# B&R Automation Studio project Model-repo
Automation Studio 4.5.2.102

## Configuration PLC

CPU X20CP1586, AutomationRuntime G4.53, Build 4.1.2, Vc V4.52.0

### Hardware
```
X20CP1586 : X20CP1586 v1.5.0.0
  Connector IF2:
    ActivateDevice = 1
    Mode = Manual
    InternetAddress = 192.168.0.5
    SubnetMask = 255.255.255.0
  Connector IF3:
    Operation = EthOnly
  ConfigurationID = JS_PLC
  ActivateOpcUa = 1
  OpcUaActivateAuditEvents = 1
  OpcUa_AuthenticationSecurityPolicy_EnableNone = 1
  OpcUa_AuthenticationSecurityPolicy_EnableBasic128Rsa15 = 1
  OpcUaInformationModels_PV_Version = 1
```

## Logical view

### Program Logical/Model/pend_mod

#### pend_mod.c
```c
/********************************************************************
 * COPYRIGHT -- Bernecker + Rainer Industrie-Elektronik Ges.m.b.H.
 ********************************************************************
 * Program: pend_mod_nlin
 * File: pend_mod.c
 * Author: Bernecker + Rainer Industrie Elektronik Ges.m.b.H.
 * Created: Fri Apr 16 22:40:22 2010
 ********************************************************************
 * Implementation of program pend_mod_nlin
 ********************************************************************
 * Generated with B&R Automation Studio Target for Simulink  V6.1.0
 * (ERT based)
 ********************************************************************/

#define _ASMATH_
#define ASMATH_
#define _ASMATH_H
#define ASMATH_H
#define _ASMATH_H_
#define ASMATH_H_
#define _ASSTRING_
#define ASSTRING_
#define _ASSTRING_H
#define ASSTRING_H
#define _ASSTRING_H_
#define ASSTRING_H_
#include <bur/plctypes.h>
#ifdef _DEFAULT_INCLUDES
#include <AsDefault.h>
#endif

#include "pend_mod_nlin.h"
#include "rtwtypes.h"

/*  Defines */

/*  Data Types */

/**************************** GLOBAL DATA *************************************/
/*  Definitions */

/*  Declarations  */

/***************************** FILE SCOPE DATA ********************************/

/*************************** FUNCTIONS ****************************************/
#ifdef __cplusplus

unsigned long bur_heap_size = 6553500;

#endif

  void _INIT mainINIT(void)
{

    UDINT st_ident;
  RTInfo_typ rt_info;
  rt_info.enable = 1;
  RTInfo(&rt_info);
  if (rt_info.cycle_time != 10000) {
    /* cycle time does not match Simulink fixed-step size */
    ST_ident("pend_mod", 0, &st_ident);
    ST_tmp_suspend(st_ident);
    ERR_warning(33310, 0);
  }

  /* initialize model */
  pend_mod_nlin_initialize();

} void _CYCLIC mainCYCLIC(void)
{
	if(start)
	{/* call model step function */
		pend_mod_nlin_output();
		pend_mod_nlin_update();
	}
	if(reset)
	{
		start = 0;
		pend_mod_nlin_initialize();
		ref = 0;
		x[0] = x[1] = x[2] = x[3] = 0;
		y[0] = y[1] = 0;
		F = 0;
		reset = 0;
	}
}  void _EXIT mainEXIT(void)
{
  /* terminate model */
  pend_mod_nlin_terminate();

} /*****************************************************************************
     Task sample time: 0.01s
   *****************************************************************************/
/*****************************************************************************
   B&R Automation Studio Target for Simulink Version: V6.1.0 (06-Nov-2019)
 *****************************************************************************/

/*======================== TOOL VERSION INFORMATION ==========================*
 * MATLAB 9.7 (R2019b)18-Jul-2019                                             *
 * Simulink 10.0 (R2019b)18-Jul-2019                                          *
 * Simulink Coder 9.2 (R2019b)18-Jul-2019                                     *
 * Embedded Coder 7.3 (R2019b)18-Jul-2019                                     *
 * Stateflow 10.1 (R2019b)18-Jul-2019                                         *
 * Fixed-Point Designer 6.4 (R2019b)18-Jul-2019                               *
 *============================================================================*/

/*======================= LICENSE IN USE INFORMATION =========================*
 * control_toolbox                                                            *
 * matlab                                                                     *
 * matlab_coder                                                               *
 * real-time_workshop                                                         *
 * rtw_embedded_coder                                                         *
 * simulink                                                                   *
 *============================================================================*/
```

### Program Logical/Controller/pend_ctrl

#### pend_ctrl_lin.h
```c
/********************************************************************
 * COPYRIGHT -- Bernecker + Rainer Industrie-Elektronik Ges.m.b.H.
 ********************************************************************
 * Program: pend_ctrl_lin
 * File: pend_ctrl_lin.h
 * Author: Bernecker + Rainer Industrie Elektronik Ges.m.b.H.
 * Created: Wed Mar 17 14:21:47 2010
 ********************************************************************
 * Header for program pend_ctrl_lin
 ********************************************************************
 * Generated with B&R Automation Studio Target for Simulink  V6.1.0
 * (ERT based)
 ********************************************************************/

#ifndef RTW_HEADER_pend_ctrl_lin_h_
#define RTW_HEADER_pend_ctrl_lin_h_
#ifndef pend_ctrl_lin_COMMON_INCLUDES_
# define pend_ctrl_lin_COMMON_INCLUDES_
#include "rtwtypes.h"
#include "rtw_continuous.h"
#include "rtw_solver.h"
#endif                                 /* pend_ctrl_lin_COMMON_INCLUDES_ */

#include <bur/plctypes.h>

#ifdef _DEFAULT_INCLUDES
 #include <AsDefault.h>
#endif

#ifndef AST_ROUND
#define AST_ROUND(x) ((x)>=0?(long long)((x)+0.5):(long long)((x)-0.5))
#endif

#include "pend_ctrl_lin_types.h"

/* Macros for accessing real-time model data structure */
#ifndef rtmGetErrorStatus
# define rtmGetErrorStatus(rtm)        ((rtm)->errorStatus)
#endif

#ifndef rtmSetErrorStatus
# define rtmSetErrorStatus(rtm, val)   ((rtm)->errorStatus = (val))
#endif

#ifndef MIN
#define MIN(a,b)                       ((a) < (b) ? (a) : (b))
#endif

#ifndef MAX
#define MAX(a,b)                       ((a) > (b) ? (a) : (b))
#endif

/* Block signals (default storage) */
typedef struct {
  real_T Input;                        /* '<S1>/Input' */
  real_T ref;                          /* '<Root>/ref' */
  real_T FeedForward;                  /* '<S4>/Feed-Forward' */
  real_T Input_f[4];                   /* '<S3>/Input' */
  real_T LQRController;                /* '<S4>/LQR Controller' */
  real_T Sum;                          /* '<S4>/Sum' */
  real_T Input1[2];                    /* '<S3>/Input1' */
} BlockIO_pend_ctrl_lin;

/* Real-time Model Data Structure */
struct tag_RTM_pend_ctrl_lin {
  const char_T *errorStatus;
};

/* Block signals (default storage) */
extern BlockIO_pend_ctrl_lin pend_ctrl_lin_B;

/* Model entry point functions */
extern void pend_ctrl_lin_initialize(void);
extern void pend_ctrl_lin_output(void);
extern void pend_ctrl_lin_update(void);
extern void pend_ctrl_lin_terminate(void);

/* Real-time Model object */
extern RT_MODEL_pend_ctrl_lin *const pend_ctrl_lin_M;

/*-
 * The generated code includes comments that allow you to trace directly
 * back to the appropriate location in the model.  The basic format
 * is <system>/block_name, where system is the system number (uniquely
 * assigned by Simulink) and block_name is the name of the block.
 *
 * Use the MATLAB hilite_system command to trace the generated code back
 * to the model.  For example,
 *
 * hilite_system('<S3>')    - opens system 3
 * hilite_system('<S3>/Kp') - opens and selects block Kp which resides in S3
 *
 * Here is the system hierarchy for this model
 *
 * '<Root>' : 'pend_ctrl_lin'
 * '<S1>'   : 'pend_ctrl_lin/B&R reference input'
 * '<S2>'   : 'pend_ctrl_lin/Configurable Controller  Subsystem1'
 * '<S3>'   : 'pend_ctrl_lin/inverted_pendulum_IOs'
 * '<S4>'   : 'pend_ctrl_lin/Configurable Controller  Subsystem1/State Feedback Controller (blks)'
 */
#endif                                 /* RTW_HEADER_pend_ctrl_lin_h_ */
```

#### pend_ctrl.c
```c
/********************************************************************
 * COPYRIGHT -- Bernecker + Rainer Industrie-Elektronik Ges.m.b.H.
 ********************************************************************
 * Program: pend_ctrl_lin
 * File: pend_ctrl.c
 * Author: Bernecker + Rainer Industrie Elektronik Ges.m.b.H.
 * Created: Wed Mar 17 14:21:47 2010
 ********************************************************************
 * Implementation of program pend_ctrl_lin
 ********************************************************************
 * Generated with B&R Automation Studio Target for Simulink  V6.1.0
 * (ERT based)
 ********************************************************************/

#define _ASMATH_
#define ASMATH_
#define _ASMATH_H
#define ASMATH_H
#define _ASMATH_H_
#define ASMATH_H_
#define _ASSTRING_
#define ASSTRING_
#define _ASSTRING_H
#define ASSTRING_H
#define _ASSTRING_H_
#define ASSTRING_H_
#include <bur/plctypes.h>
#ifdef _DEFAULT_INCLUDES
#include <AsDefault.h>
#endif

#include "pend_ctrl_lin.h"
#include "rtwtypes.h"

/*  Defines */

/*  Data Types */

/**************************** GLOBAL DATA *************************************/
/*  Definitions */

/*  Declarations  */

/***************************** FILE SCOPE DATA ********************************/

/*************************** FUNCTIONS ****************************************/
#ifdef __cplusplus

unsigned long bur_heap_size = 6553500;

#endif

  void _INIT mainINIT(void)
{

    UDINT st_ident;
  RTInfo_typ rt_info;
  rt_info.enable = 1;
  RTInfo(&rt_info);
  if (rt_info.cycle_time != 10000) {
    /* cycle time does not match Simulink fixed-step size */
    ST_ident("pend_ctrl", 0, &st_ident);
    ST_tmp_suspend(st_ident);
    ERR_warning(33310, 0);
  }

  /* initialize model */
  pend_ctrl_lin_initialize();

} void _CYCLIC mainCYCLIC(void)
{
  /* call model step function */
  pend_ctrl_lin_output();

  pend_ctrl_lin_update();

} void _EXIT mainEXIT(void)
{
  /* terminate model */
  pend_ctrl_lin_terminate();

} /*****************************************************************************
     Task sample time: 0.01s
   *****************************************************************************/
/*****************************************************************************
   B&R Automation Studio Target for Simulink Version: V6.1.0 (06-Nov-2019)
 *****************************************************************************/

/*======================== TOOL VERSION INFORMATION ==========================*
 * MATLAB 9.7 (R2019b)18-Jul-2019                                             *
 * Simulink 10.0 (R2019b)18-Jul-2019                                          *
 * Simulink Coder 9.2 (R2019b)18-Jul-2019                                     *
 * Embedded Coder 7.3 (R2019b)18-Jul-2019                                     *
 * Stateflow 10.1 (R2019b)18-Jul-2019                                         *
 * Fixed-Point Designer 6.4 (R2019b)18-Jul-2019                               *
 *============================================================================*/

/*======================= LICENSE IN USE INFORMATION =========================*
 * control_toolbox                                                            *
 * matlab                                                                     *
 * matlab_coder                                                               *
 * real-time_workshop                                                         *
 * rtw_embedded_coder                                                         *
 * simulink                                                                   *
 *============================================================================*/
```

#### pend_ctrl_lin.c
```c
/********************************************************************
 * COPYRIGHT -- Bernecker + Rainer Industrie-Elektronik Ges.m.b.H.
 ********************************************************************
 * Program: pend_ctrl_lin
 * File: pend_ctrl_lin.c
 * Author: Bernecker + Rainer Industrie Elektronik Ges.m.b.H.
 * Created: Wed Mar 17 14:21:47 2010
 ********************************************************************
 * Implementation of program pend_ctrl_lin
 ********************************************************************
 * Generated with B&R Automation Studio Target for Simulink  V6.1.0
 * (ERT based)
 ********************************************************************/

#include "pend_ctrl_lin.h"
#include "pend_ctrl_lin_private.h"

/*  Defines */

/*  Data Types */

/**************************** GLOBAL DATA *************************************/
/*  Definitions */

/* Block signals (default storage) */
BlockIO_pend_ctrl_lin pend_ctrl_lin_B;

/* Real-time model */
RT_MODEL_pend_ctrl_lin pend_ctrl_lin_M_;
RT_MODEL_pend_ctrl_lin *const pend_ctrl_lin_M = &pend_ctrl_lin_M_;

/*  Declarations  */

/***************************** FILE SCOPE DATA ********************************/

/*************************** FUNCTIONS ****************************************/

/* Model output function */
void pend_ctrl_lin_output(void)
{
  real_T tmp;

  /* S-Function (bur_in): '<S1>/Input' */
  pend_ctrl_lin_B.Input = ref;

  /* Gain: '<Root>/ref' */
  pend_ctrl_lin_B.ref = 10.0 * pend_ctrl_lin_B.Input;

  /* Gain: '<S4>/Feed-Forward' */
  pend_ctrl_lin_B.FeedForward = -2987.4616903679112 * pend_ctrl_lin_B.ref;

  /* S-Function (bur_in): '<S3>/Input' */
  pend_ctrl_lin_B.Input_f[0] = x[0];
  pend_ctrl_lin_B.Input_f[1] = x[1];
  pend_ctrl_lin_B.Input_f[2] = x[2];
  pend_ctrl_lin_B.Input_f[3] = x[3];

  /* Gain: '<S4>/LQR Controller' */
  tmp = -2987.4616903679125 * pend_ctrl_lin_B.Input_f[0];
  tmp += -3740.1178916812455 * pend_ctrl_lin_B.Input_f[1];
  tmp += -32774.860875805127 * pend_ctrl_lin_B.Input_f[2];
  tmp += -7399.4348019785593 * pend_ctrl_lin_B.Input_f[3];
  pend_ctrl_lin_B.LQRController = tmp;

  /* Sum: '<S4>/Sum' */
  pend_ctrl_lin_B.Sum = pend_ctrl_lin_B.FeedForward -
    pend_ctrl_lin_B.LQRController;

  /* S-Function (bur_in): '<S3>/Input1' */
  pend_ctrl_lin_B.Input1[0] = y[0];
  pend_ctrl_lin_B.Input1[1] = y[1];

  /* S-Function (bur_out): '<S3>/Output' */
  F = pend_ctrl_lin_B.Sum;
}

/* Model update function */
void pend_ctrl_lin_update(void)
{
  /* (no update code required) */
}

/* Model initialize function */
void pend_ctrl_lin_initialize(void)
{
  /* (no initialization code required) */
}

/* Model terminate function */
void pend_ctrl_lin_terminate(void)
{
  /* (no terminate code required) */
}

/*======================== TOOL VERSION INFORMATION ==========================*
 * MATLAB 9.7 (R2019b)18-Jul-2019                                             *
 * Simulink 10.0 (R2019b)18-Jul-2019                                          *
 * Simulink Coder 9.2 (R2019b)18-Jul-2019                                     *
 * Embedded Coder 7.3 (R2019b)18-Jul-2019                                     *
 * Stateflow 10.1 (R2019b)18-Jul-2019                                         *
 * Fixed-Point Designer 6.4 (R2019b)18-Jul-2019                               *
 *============================================================================*/

/*======================= LICENSE IN USE INFORMATION =========================*
 * control_toolbox                                                            *
 * matlab                                                                     *
 * matlab_coder                                                               *
 * real-time_workshop                                                         *
 * rtw_embedded_coder                                                         *
 * simulink                                                                   *
 *============================================================================*/
```

### Global.var - Global variables of pend_ctrl
```iecst
VAR
	reset : BOOL := FALSE;
	ref : LREAL := 0; (*Reference input*)
	x : ARRAY[0..3] OF LREAL := [4(0)]; (*Inverted pendulum state x*)
	y : ARRAY[0..1] OF LREAL := [2(0)]; (*Inverted pendulum output y*)
	F : LREAL := 0; (*Car force*)
	start : BOOL := FALSE;
END_VAR
```

Listed in the project but not available here: Logical/Libraries, Logical/MATLAB_includes, Logical/Global.typ
